ABB RAPID module: movement

MODULE movement
    PERS string action;
    PERS robjoint joints;
    PERS speeddata speed;
    PERS num jogdir{3};
    PERS num joggingjoints{6};
    PERS robtarget target_pos;
    PROC Main()
        WHILE TRUE DO
            ! Continuously see what is required to be done, if the server sets an action then perform that action.
            TEST action
            CASE "MJ":
                MoveAbsJ [joints,[9e9,9e9,9e9,9e9,9e9,9e9]], speed, fine, tSCup;
            CASE "JL":
                joglinear;
            CASE "JJ":
                jogjoint;
            CASE "PA":
                StorePath;
                StopMove;
            CASE "RE":
                RestoPath;
                StartMove;
            CASE "ST":
                StopMove;
                ClearPath;
                joggingjoints := [0,0,0,0,0,0];
                joints := [0,0,0,0,0,0];
            CASE "MC":
                MoveL target_pos, speed, fine, tSCup;
            CASE "MT":
                MoveL target_pos, speed, fine, tSCup;
            IF action <> "L" AND action <> "J" AND action <> "A" THEN
                action := "";
            ENDIF
            ENDTEST
        ENDWHILE
    ENDPROC

    PROC joglinear()
        ! this function reads in persistent variables and then sets the robot target to be slightly further away in the requested direction
        ! than the current target
        var robtarget curr_target;
        curr_target := CRobT(\Tool:=tSCup);
        MoveL Offs(curr_target, jogdir{1}*100, jogdir{2}*100, jogdir{3}*100), speed, fine, tSCup;
    ENDPROC

    PROC jogjoint()
        !this function reads in persistent variables and then sets the robot target to be slightly further away in the requested angles
        ! than the current target
        VAR jointtarget jointsout;
        jointsout := CJointT();
        jointsout.robax.rax_1 := jointsout.robax.rax_1 + joggingjoints{1};
        jointsout.robax.rax_2 := jointsout.robax.rax_2 + joggingjoints{1};
        jointsout.robax.rax_3 := jointsout.robax.rax_3 + joggingjoints{1};
        jointsout.robax.rax_4 := jointsout.robax.rax_4 + joggingjoints{1};
        jointsout.robax.rax_5 := jointsout.robax.rax_5 + joggingjoints{1};
        jointsout.robax.rax_6 := jointsout.robax.rax_6 + joggingjoints{1};

        MoveAbsJ jointsout, speed, fine, tSCup;
    ENDPROC
ENDMODULE
